PROGRAM MAIN
VAR
	StartButton: BOOL;
	LineRun: BOOL;
	StopButton: BOOL;
	BoxConveyorRun: BOOL;
	AppleConveyorRun: BOOL;
	ctuParts: CTU;
	ApplePresent: BOOL;
	BoxPresent: BOOL;
END_VAR

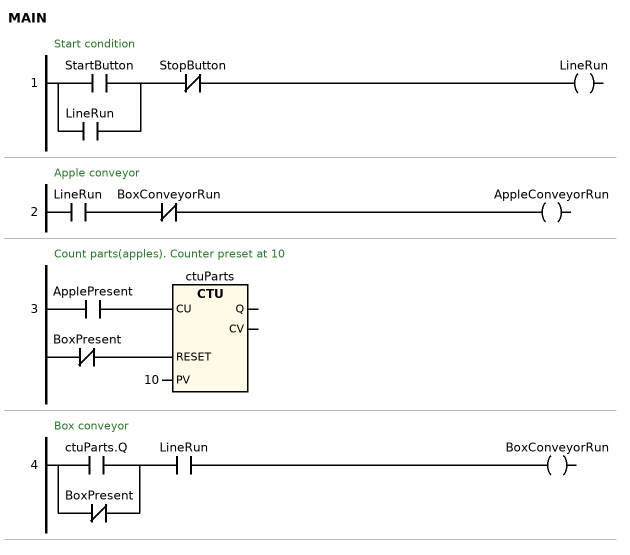
// NETWORK 1
// Start condition
LineRun := (StartButton OR LineRun) AND NOT StopButton;

// NETWORK 2
// Apple conveyor
AppleConveyorRun := LineRun AND NOT BoxConveyorRun;

// NETWORK 3
// Count parts(apples). Counter preset at 10
ctuParts(CU := ApplePresent, RESET := NOT BoxPresent, PV := 10); // CTU

// NETWORK 4
// Box conveyor
BoxConveyorRun := (ctuParts.Q OR NOT BoxPresent) AND LineRun;

END_PROGRAM

(* stored: Version 1.1.0.1, ProductVersion 3.1.4024.15
   POU MAIN: Id {8301d6fd-d90a-41a6-816f-08c3e5233f51}, SpecialFunc None *)
